TYPE ST_PneumaticPressParCmd :
STRUCT
    Reserved : BOOL;
END_STRUCT
END_TYPE

(* stored: Version 1.1.0.1, ProductVersion 3.1.4024.12
   DUT ST_PneumaticPressParCmd: Id {0ccaa7cf-48a7-4b25-94d9-29e3b8830c14} *)
